% RSLogix 500 project PRACTISE-8.2.RSS, saved by version 8.30.00.16 %
PROJECT "UNTITLED"    % processor: MicroLogix 1000 %

PROGRAM FILES
  LAD 2 "MAIN_PROG"  18 rungs
  LAD 3 "USER_FAULT"  1 rungs
  LAD 4 "HSC_INT"  1 rungs
  LAD 5 "STI_INT"  1 rungs
  LAD 6, 7, 8, 9, 10, 11, 12, 13, 14, 15, 16: only END

DATA FILES
  O0 OUTPUT  1 elements
  I1 INPUT  2 elements
  S2 STATUS  33 elements
  B3 BINARY  32 elements
  T4 TIMER  40 elements
  C5 COUNTER  32 elements
  R6 CONTROL  16 elements
  N7 INTEGER  105 elements

LADDER 2 "MAIN_PROG"
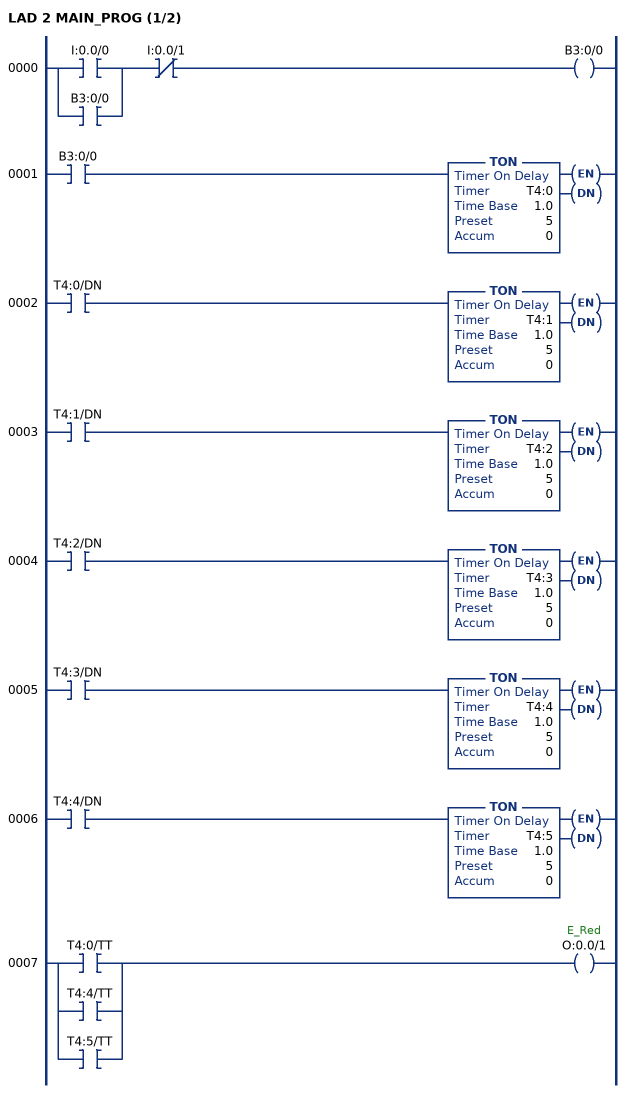
% Rung: 0 %
SOR BST XIC I:0.0/0 NXB XIC B3:0/0 BND XIO I:0.0/1 OTE B3:0/0 EOR
% Rung: 1 %
SOR XIC B3:0/0 TON T4:0 1.0 5 0 EOR
% Rung: 2 %
SOR XIC T4:0/DN TON T4:1 1.0 5 0 EOR
% Rung: 3 %
SOR XIC T4:1/DN TON T4:2 1.0 5 0 EOR
% Rung: 4 %
SOR XIC T4:2/DN TON T4:3 1.0 5 0 EOR
% Rung: 5 %
SOR XIC T4:3/DN TON T4:4 1.0 5 0 EOR
% Rung: 6 %
SOR XIC T4:4/DN TON T4:5 1.0 5 0 EOR
% Rung: 7 %
SOR BST XIC T4:0/TT NXB BST XIC T4:4/TT NXB XIC T4:5/TT BND BND OTE O:0.0/1 EOR
%   O:0.0/1  "E_Red" %

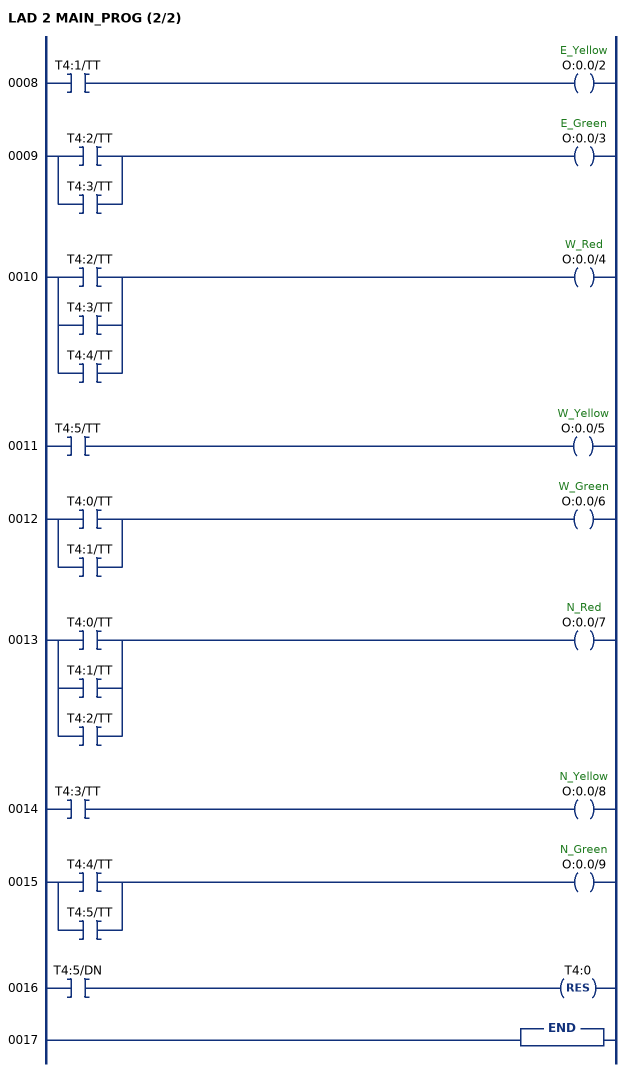
% Rung: 8 %
SOR XIC T4:1/TT OTE O:0.0/2 EOR
%   O:0.0/2  "E_Yellow" %
% Rung: 9 %
SOR BST XIC T4:2/TT NXB XIC T4:3/TT BND OTE O:0.0/3 EOR
%   O:0.0/3  "E_Green" %
% Rung: 10 %
SOR BST XIC T4:2/TT NXB BST XIC T4:3/TT NXB XIC T4:4/TT BND BND OTE O:0.0/4 EOR
%   O:0.0/4  "W_Red" %
% Rung: 11 %
SOR XIC T4:5/TT OTE O:0.0/5 EOR
%   O:0.0/5  "W_Yellow" %
% Rung: 12 %
SOR BST XIC T4:0/TT NXB XIC T4:1/TT BND OTE O:0.0/6 EOR
%   O:0.0/6  "W_Green" %
% Rung: 13 %
SOR BST XIC T4:0/TT NXB BST XIC T4:1/TT NXB XIC T4:2/TT BND BND OTE O:0.0/7 EOR
%   O:0.0/7  "N_Red" %
% Rung: 14 %
SOR XIC T4:3/TT OTE O:0.0/8 EOR
%   O:0.0/8  "N_Yellow" %
% Rung: 15 %
SOR BST XIC T4:4/TT NXB XIC T4:5/TT BND OTE O:0.0/9 EOR
%   O:0.0/9  "N_Green" %
% Rung: 16 %
SOR XIC T4:5/DN RES T4:0 EOR
% Rung: 17 %
SOR END EOR

DATA TABLE (non-zero values as saved)
DATA T4
% .PRE .ACC %
% T4:0 % 5 0
% T4:1 % 5 0
% T4:2 % 5 0
% T4:3 % 5 0
% T4:4 % 5 0
% T4:5 % 5 0
